// TwinCAT 3 PLC project PickPlacePlc
// ProgramVersion: 3.1.4026.25
// libraries:
//   Tc2_Standard, * (Beckhoff Automation GmbH)
//   Tc2_System, * (Beckhoff Automation GmbH)
// project tree:
//   / PlcTask.TcTTO
//   Framework/ I_Node.TcIO, E_OpMode.TcDUT, E_CmdResult.TcDUT, GVL_Framework.TcGVL, FB_CyclicNode.TcPOU, FB_ModeNode.TcPOU, FB_CycleManager.TcPOU, FB_OpModeHandler.TcPOU
//   Devices/ FB_PneumaticCylinder.TcPOU
//   Machine/ FB_HandlingUnit.TcPOU, FB_Machine.TcPOU, MAIN.TcPOU
// real-time tasks:
//   TASK PlcTask: cycle T#10ms, priority 20, ADS port 350

CONFIGURATION PickPlacePlc
    RESOURCE PLC ON TwinCAT3
        TASK PlcTask(INTERVAL := T#10ms, PRIORITY := 20);
        PROGRAM MAIN WITH PlcTask : MAIN;
    END_RESOURCE
END_CONFIGURATION

// ---- Framework/E_OpMode.TcDUT
{attribute 'qualified_only'}
{attribute 'strict'}
TYPE E_OpMode :
(
    eStop      := 0,   // machine halted / safe
    eManual    := 1,   // operator jogs single devices from the HMI
    eHoming    := 2,   // move every node to its defined home position
    eAutomatic := 3    // run the production sequences
) DINT;
END_TYPE

// ---- Framework/E_CmdResult.TcDUT
{attribute 'qualified_only'}
{attribute 'strict'}
TYPE E_CmdResult :
(
    eBusy  := 0,   // command still running, keep calling it
    eDone  := 1,   // command finished successfully -> advance the step
    eError := 2    // command failed (e.g. move timeout) -> handle the error
) DINT;
END_TYPE

// ---- Framework/GVL_Framework.TcGVL
{attribute 'qualified_only'}
VAR_GLOBAL CONSTANT
    // Max direct children a single node may register.
    // Bumped only if a real machine node grows very wide.
    cMaxChildren : DINT := 16;
END_VAR

// ---- Framework/I_Node.TcIO
// I_Node - the one thing every element in the machine tree can do.
// The whole framework talks to nodes only through this interface, which is
// why a generic parent can hold a mixed list of devices and mode nodes.
INTERFACE I_Node

// Run this node once, then recurse into its children.
METHOD Cyclic
VAR_INPUT
END_VAR
END_METHOD

METHOD RegisterChild
VAR_INPUT
    ipChild : I_Node;   // child that wants to join this node in the tree
END_VAR
END_METHOD

METHOD SetMode
VAR_INPUT
    eNewMode : E_OpMode;   // pushed down the tree by the OpModeHandler
END_VAR
END_METHOD

END_INTERFACE

// ---- Machine/MAIN.TcPOU
// MAIN - the whole application is three declarations and two calls.
//
// fbMachine is the root of the node tree (ipParent := 0 -> no parent).
// Declaring it constructs the entire tree, because every child registered
// itself with its parent during FB_init.
PROGRAM MAIN
VAR
    fbMachine : FB_Machine(ipParent := 0, sNodeName := 'Machine');
    fbOpMode  : FB_OpModeHandler;
    bInit     : BOOL := TRUE;
END_VAR

// First-scan wiring: tell the op-mode handler which node is the root.
IF bInit THEN
    fbOpMode.SetRoot(fbMachine);
    fbOpMode.Mode := E_OpMode.eAutomatic;   // demo: start running immediately
    bInit := FALSE;
END_IF

// One call runs the whole machine: mode is pushed down, then the tree ticks.
fbOpMode.Cyclic();

END_PROGRAM

// ---- Machine/FB_Machine.TcPOU
// FB_Machine - the root node of the tree.
//
// It holds the top-level functional units (here just one handling unit). Its
// own RunAutomatic stays empty: each unit runs its own sequence via the tree.
// This is where you would add machine-wide coordination between units later.
FUNCTION_BLOCK FB_Machine EXTENDS FB_ModeNode
VAR
    fbHandling : FB_HandlingUnit(ipParent := THIS^, sNodeName := 'HandlingUnit');
END_VAR

METHOD PROTECTED RunAutomatic
VAR_INPUT
END_VAR
// No machine-level coordination needed for a single unit.
;
END_METHOD

END_FUNCTION_BLOCK

// ---- Framework/FB_ModeNode.TcPOU
// FB_ModeNode - a functional unit that owns process logic (cinnamon's
// CNM_AbstractModeNode). It is still a cyclic node, but its per-cycle work is
// dispatched to one method per operating mode. A derived unit only implements
// the modes it cares about (RunAutomatic is mandatory; the rest default to
// doing nothing).
FUNCTION_BLOCK ABSTRACT FB_ModeNode EXTENDS FB_CyclicNode
VAR
    // (no own variables - state lives in the concrete unit)
END_VAR

// Override of FB_CyclicNode.OnCyclic: route the cycle by current op-mode.
METHOD PROTECTED OnCyclic
VAR_INPUT
END_VAR
CASE eMode OF
    E_OpMode.eManual:    THIS^.RunManual();
    E_OpMode.eHoming:    THIS^.RunHoming();
    E_OpMode.eAutomatic: THIS^.RunAutomatic();
ELSE
    THIS^.RunStop();     // eStop and anything unexpected
END_CASE
END_METHOD

// Production sequence. Every mode node must implement this.
METHOD PROTECTED ABSTRACT RunAutomatic
VAR_INPUT
END_VAR
END_METHOD

// Default: nothing. Override to allow operator jogging.
METHOD PROTECTED RunManual
VAR_INPUT
END_VAR
END_METHOD

// Default: nothing. Override to move the unit to its home position.
METHOD PROTECTED RunHoming
VAR_INPUT
END_VAR
END_METHOD

// Default: nothing. Override to park the unit safely on stop.
METHOD PROTECTED RunStop
VAR_INPUT
END_VAR
END_METHOD

END_FUNCTION_BLOCK

// ---- Framework/FB_CyclicNode.TcPOU
// FB_CyclicNode - the base of every element in the machine.
//
// This is the counterpart of cinnamon's CNM_AbstractCyclicNode: a "device" or
// monitored component that gets called every cycle. It owns a list of children
// and, via FB_init, registers itself with its parent. That is the whole
// hierarchical-composition trick: build the tree by declaration, and one call
// on the root fans out to everything.
//
// ABSTRACT: OnCyclic is not implemented here, so this FB cannot be instantiated
// directly. Concrete devices (e.g. FB_PneumaticCylinder) override OnCyclic.
FUNCTION_BLOCK ABSTRACT FB_CyclicNode IMPLEMENTS I_Node
VAR
    sName       : STRING;                                 // node name (also its HMI/log label)
    eMode       : E_OpMode;                               // current op-mode, pushed down from the root
    aChildren   : ARRAY[1..GVL_Framework.cMaxChildren] OF I_Node;
    nChildCount : DINT;
END_VAR

METHOD FB_init : BOOL
VAR_INPUT
    bInitRetains : BOOL;    // TwinCAT-supplied
    bInCopyCode  : BOOL;    // TwinCAT-supplied
    ipParent     : I_Node;  // pass THIS^ of the parent, or 0 for the root
    sNodeName    : STRING;  // human-readable name of this node
END_VAR
sName := sNodeName;
// A node registers itself with its parent the moment it is declared.
IF ipParent <> 0 THEN
    ipParent.RegisterChild(THIS^);
END_IF
END_METHOD

METHOD PUBLIC RegisterChild
VAR_INPUT
    ipChild : I_Node;
END_VAR
IF ipChild <> 0 AND_THEN nChildCount < GVL_Framework.cMaxChildren THEN
    nChildCount := nChildCount + 1;
    aChildren[nChildCount] := ipChild;
END_IF
END_METHOD

METHOD PUBLIC Cyclic
VAR
    nI : DINT;
END_VAR
// Run this node first (set targets / drive I/O), then let the children act.
THIS^.OnCyclic();
FOR nI := 1 TO nChildCount DO
    aChildren[nI].Cyclic();
END_FOR
END_METHOD

METHOD PUBLIC SetMode
VAR_INPUT
    eNewMode : E_OpMode;
END_VAR
VAR
    nI : DINT;
END_VAR
eMode := eNewMode;
FOR nI := 1 TO nChildCount DO
    aChildren[nI].SetMode(eNewMode);
END_FOR
END_METHOD

// The node's own per-cycle work. Implemented by every concrete node.
METHOD PROTECTED ABSTRACT OnCyclic
VAR_INPUT
END_VAR
END_METHOD

END_FUNCTION_BLOCK

// ---- Machine/FB_HandlingUnit.TcPOU
// FB_HandlingUnit - a functional unit with real process logic.
//
// It owns two devices (a lift cylinder and a gripper) and drives a full
// pick-and-place cycle through the CycleManager. Note how the children are
// declared with (ipParent := THIS^, ...): that single line is what puts them
// under this unit in the tree - no wiring, no registration call.
FUNCTION_BLOCK FB_HandlingUnit EXTENDS FB_ModeNode
VAR
    fbLift    : FB_PneumaticCylinder(ipParent := THIS^, sNodeName := 'Lift');
    fbGripper : FB_PneumaticCylinder(ipParent := THIS^, sNodeName := 'Gripper');
    fbCycle   : FB_CycleManager;
END_VAR

METHOD PROTECTED RunAutomatic
VAR_INPUT
END_VAR
// One pick-and-place loop. Await() advances the step as each command reports
// eDone; when the last step finishes, Restart() loops the cycle.
fbCycle.Call(bExecute := TRUE);

CASE fbCycle.Step OF
    0: fbCycle.Await(fbGripper.Retract());  // make sure the gripper is open
    1: fbCycle.Await(fbLift.Extend());      // lower onto the part
    2: fbCycle.Await(fbGripper.Extend());   // close gripper (pick)
    3: fbCycle.Await(fbLift.Retract());     // lift the part
    4: fbCycle.Await(fbLift.Extend());      // lower at the place position
    5: fbCycle.Await(fbGripper.Retract());  // open gripper (place)
    6: fbCycle.Await(fbLift.Retract());     // lift clear
ELSE
    fbCycle.Restart();                      // cycle complete -> run it again
END_CASE
END_METHOD

METHOD PROTECTED RunStop
VAR_INPUT
END_VAR
// Leaving automatic: reset the step engine so the next start begins at step 0.
fbCycle.Reset();
END_METHOD

END_FUNCTION_BLOCK

// ---- Devices/FB_PneumaticCylinder.TcPOU
// FB_PneumaticCylinder - a reusable device driver (a leaf node in the tree).
//
// This is the cinnamon idea of a hardware driver: the outside world only sees
// two commands, Extend() and Retract(), each returning an E_CmdResult. The
// device itself owns the coils, the end sensors and the move-timeout watchdog.
// The gripper in this demo is just another instance of this driver.
//
// bSimulate is on by default so the sequence steps on a soft-PLC with no I/O
// mapped: the end sensors are faked after tSimStroke. Set it FALSE and map the
// four I/O variables to real terminals for a machine.
FUNCTION_BLOCK FB_PneumaticCylinder EXTENDS FB_CyclicNode
VAR
    // --- Hardware I/O (map to real terminals; e.g. AT %Q* / AT %I*) ---
    bExtendCoil      : BOOL;
    bRetractCoil     : BOOL;
    bExtendedSensor  : BOOL;
    bRetractedSensor : BOOL;

    // --- Configuration ---
    tMoveTimeout     : TIME := T#5S;
    bSimulate        : BOOL := TRUE;
    tSimStroke       : TIME := T#500MS;

    // --- Internal state ---
    bTargetExtend    : BOOL;
    bLastTarget      : BOOL;
    fbTimeout        : TON;
    fbSimStroke      : TON;
END_VAR

// Command the cylinder out. Returns eBusy until the extended sensor is set,
// eError if the move times out, eDone when it arrives.
METHOD PUBLIC Extend : E_CmdResult
VAR_INPUT
END_VAR
bTargetExtend := TRUE;
IF bExtendedSensor THEN
    Extend := E_CmdResult.eDone;
ELSIF fbTimeout.Q THEN
    Extend := E_CmdResult.eError;
ELSE
    Extend := E_CmdResult.eBusy;
END_IF
END_METHOD

METHOD PUBLIC Retract : E_CmdResult
VAR_INPUT
END_VAR
bTargetExtend := FALSE;
IF bRetractedSensor THEN
    Retract := E_CmdResult.eDone;
ELSIF fbTimeout.Q THEN
    Retract := E_CmdResult.eError;
ELSE
    Retract := E_CmdResult.eBusy;
END_IF
END_METHOD

METHOD PROTECTED OnCyclic
VAR_INPUT
END_VAR
// Drive the coils from the target and supervise the move. Runs every cycle,
// even in steps where no command is calling this cylinder, so it holds state.
bExtendCoil  := bTargetExtend;
bRetractCoil := NOT bTargetExtend;

fbTimeout(IN := (bTargetExtend AND NOT bExtendedSensor)
              OR (NOT bTargetExtend AND NOT bRetractedSensor),
          PT := tMoveTimeout);

IF bSimulate THEN
    // On a target change, clear both sensors and restart the stroke timer.
    IF bTargetExtend <> bLastTarget THEN
        bExtendedSensor  := FALSE;
        bRetractedSensor := FALSE;
        bLastTarget      := bTargetExtend;
        fbSimStroke(IN := FALSE);
    END_IF
    fbSimStroke(IN := TRUE, PT := tSimStroke);
    IF fbSimStroke.Q THEN
        bExtendedSensor  := bTargetExtend;
        bRetractedSensor := NOT bTargetExtend;
    END_IF
END_IF
END_METHOD

END_FUNCTION_BLOCK

// ---- Framework/FB_CycleManager.TcPOU
// FB_CycleManager - the step engine (cinnamon's CNM_CycleManager, trimmed to
// the essentials). It replaces the hand-rolled "CASE nStep OF ... nStep := ..."
// pattern: you still write a CASE, but the manager owns the step counter, the
// start edge, error latching and stepping.
//
// Usage inside a RunAutomatic method:
//
//     fbCycle.Call(bExecute := TRUE);          // TRUE = run continuously
//     CASE fbCycle.Step OF
//         0: fbCycle.Await(fbLift.Extend());   // advances when the cmd is eDone
//         1: fbCycle.Await(fbGripper.Extend());
//         ...
//     END_CASE
FUNCTION_BLOCK FB_CycleManager
VAR
    nStep      : DINT;
    bActive    : BOOL;
    bError     : BOOL;
    rtrigStart : R_TRIG;
END_VAR

METHOD PUBLIC Call
VAR_INPUT
    bExecute : BOOL;   // level signal: rising edge starts at step 0
END_VAR
rtrigStart(CLK := bExecute);
IF rtrigStart.Q THEN
    nStep   := 0;
    bError  := FALSE;
    bActive := TRUE;
END_IF
IF NOT bExecute THEN
    bActive := FALSE;   // dropping execute stops the sequence
END_IF
END_METHOD

METHOD PUBLIC Await : BOOL   // TRUE on the cycle the step actually advances
VAR_INPUT
    eResult : E_CmdResult;   // result of the command evaluated in this step
END_VAR
Await := FALSE;
IF NOT bActive THEN
    RETURN;
END_IF
CASE eResult OF
    E_CmdResult.eDone:
        nStep   := nStep + 1;
        Await   := TRUE;
    E_CmdResult.eError:
        bError  := TRUE;
        bActive := FALSE;   // hold on error; caller decides what to do next
END_CASE
END_METHOD

// Jump back to step 0 and keep running (used to loop a finished cycle).
METHOD PUBLIC Restart
VAR_INPUT
END_VAR
nStep   := 0;
bError  := FALSE;
bActive := TRUE;
END_METHOD

// Full stop: also clears the start edge so re-entering a mode restarts cleanly.
METHOD PUBLIC Reset
VAR_INPUT
END_VAR
nStep   := 0;
bError  := FALSE;
bActive := FALSE;
rtrigStart(CLK := FALSE);
END_METHOD

PROPERTY PUBLIC Step : DINT
GET
Step := nStep;
END_GET
END_PROPERTY

PROPERTY PUBLIC Active : BOOL
GET
Active := bActive;
END_GET
END_PROPERTY

PROPERTY PUBLIC Error : BOOL
GET
Error := bError;
END_GET
END_PROPERTY

END_FUNCTION_BLOCK

// ---- Framework/FB_OpModeHandler.TcPOU
// FB_OpModeHandler - the single entry point MAIN calls each cycle.
// It holds the machine's operating mode, pushes it down the whole tree, then
// runs the tree. In a real project this is where you would gate mode changes
// on the safety state, latch requests from the HMI, etc.
FUNCTION_BLOCK FB_OpModeHandler
VAR
    ipRoot : I_Node;
    eMode  : E_OpMode := E_OpMode.eStop;
END_VAR

METHOD PUBLIC SetRoot
VAR_INPUT
    ipRootNode : I_Node;   // the machine node
END_VAR
ipRoot := ipRootNode;
END_METHOD

METHOD PUBLIC Cyclic
VAR_INPUT
END_VAR
IF ipRoot <> 0 THEN
    ipRoot.SetMode(eMode);   // distribute the mode to every node
    ipRoot.Cyclic();         // then run the whole tree
END_IF
END_METHOD

PROPERTY PUBLIC Mode : E_OpMode
GET
Mode := eMode;
END_GET
SET
eMode := Mode;
END_SET
END_PROPERTY

END_FUNCTION_BLOCK
